FUNCTION_BLOCK FB_AuditLogListener EXTENDS FB_CyclicFB IMPLEMENTS I_AuditLogListener

VAR
    MessageListener : FB_AuditLogMsgListener;
	
//	logger : FB_Logger;
END_VAR

METHOD CyclicLogic
IF NOT _InitComplete THEN
    _InitComplete := Initialize();
    RETURN;
END_IF

MessageListener.Execute();
END_METHOD

METHOD Initialize : BOOL
VAR
    ListenerFilter : FB_TcEventFilter;
    hr             : HRESULT;
END_VAR
MessageListener.Listener := THIS^;                                   //For callbacks on message received
ListenerFilter.Clear().EventClass.EqualTo(TC_EVENT_CLASSES.AuditLog); //Filter events by tracing class
hr := MessageListener.Subscribe2(ListenerFilter);                    //Subscribe to retrieve defined events
IF SUCCEEDED(hr) THEN
    Initialize := TRUE;
END_IF
END_METHOD

METHOD OnTraceReceived
VAR_INPUT
    message : ST_AuditLogMessages;
END_VAR

VAR
	timestamp: Tc2_System.T_MaxString;
	key: Tc2_System.T_MaxString;
	value: Tc2_System.T_MaxString;
END_VAR
// Extract relevant fields
timestamp   := message.Timestamp;
key   := message.k;
value   := message.v;
END_METHOD

END_FUNCTION_BLOCK

(* stored: Version 1.1.0.1
   POU FB_AuditLogListener: Id {75253406-65a3-47be-ae4f-01a902b48fd8}, SpecialFunc None
   Method CyclicLogic: Id {edcf0414-95ac-46d9-994d-48e42eecc40d}
   Method Initialize: Id {1ae9c531-8a99-447d-a014-f6ebbb22892c}
   Method OnTraceReceived: Id {fbc28f07-e424-409d-97b1-6ae130fcbfaf} *)
